# EPICS substitutions: db/FC_HV.substitutions
file "FC_HV.template"

{
  pattern {IOC,           MASTER_ID, SLAVE_POS, HWTYPE, CH_ID, DESC}
          {"LEBT-010:PBI-FC-001", 0,     4,       "EL3174_0to10V",   AI1,   "$(HV):Volt-RB"}
          {"LEBT-010:PBI-FC-001", 0,     4,       "EL3174_0to10V",   AI2,   "$(HV):Curr-RB"}
          {"LEBT-010:PBI-FC-001", 0,     5,       "EL4134",   AO1,   "$(HV):Volt"}
          {"LEBT-010:PBI-FC-001", 0,     5,	  "EL4134",   AO1-RB,"$(HV):Volt-RB"}
          {"LEBT-010:PBI-FC-001", 0,     5,       "EL4134",   AO2,   "$(HV):Curr"}
          {"LEBT-010:PBI-FC-001", 0,     5,	  "EL4134",   AO2-RB,"$(HV):Curr-RB"}
          {"LEBT-010:PBI-FC-001", 0,     7,	  "EL2124",   BO2,   "$(HV):Pol"}
          {"LEBT-010:PBI-FC-001", 0,     7,       "EL2124",   BO2-RB,"$(HV):Pol-RB"}
          {"LEBT-010:PBI-FC-001", 0,     7,	  "EL2124",   BO1,   "$(HV):Bias"}
          {"LEBT-010:PBI-FC-001", 0,     7,       "EL2124",   BO1-RB,"$(HV):Bias-RB"}
}
